Yaskawa INFORM job: FIGURE.JBI

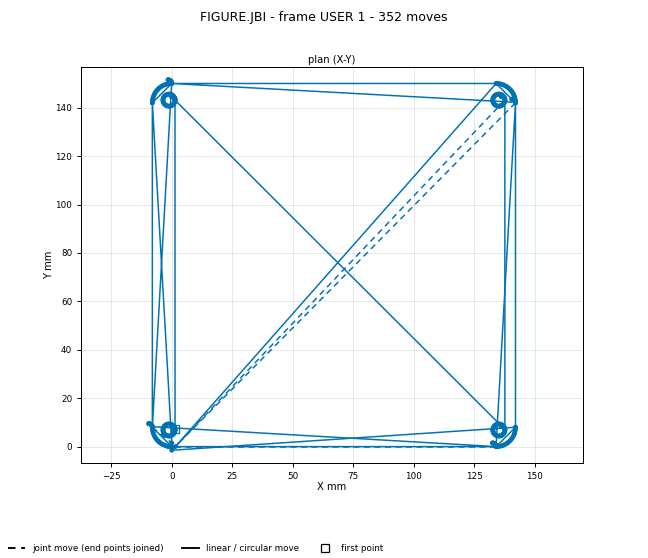
[picture p0: tool path of FIGURE.JBI in frame USER 1, 352 of 352 moves have a stored position in this frame; points joined in program order, loops and branches not executed]
/JOB
//NAME FIGURE
//POS
///NPOS 352,0,0,0,0,0
///TOOL 1
///USER 1
///POSTYPE USER
///RECTAN
///RCONF 1,0,0,0,0,0,0,0,0,0,0,0,0,0,0,0,0,0,0,0,0,0,0,0
C00000=1.357,7.11,7.0,0,0,0
C00001=1.302,7.339,7.0,0,0,0
C00002=1.212,7.556,7.0,0,0,0
C00003=1.089,7.757,7.0,0,0,0
C00004=0.936,7.936,7.0,0,0,0
C00005=0.757,8.089,7.0,0,0,0
C00006=0.556,8.212,7.0,0,0,0
C00007=0.339,8.302,7.0,0,0,0
C00008=0.11,8.357,7.0,0,0,0
C00009=-0.125,8.375,7.0,0,0,0
C00010=-0.125,8.375,7.0,0,0,0
C00011=1.375,6.875,7.0,0,0,0
C00012=1.344,7.266,7.0,0,0,0
C00013=1.253,7.648,7.0,0,0,0
C00014=1.103,8.01,7.0,0,0,0
C00015=0.898,8.344,7.0,0,0,0
C00016=0.643,8.643,7.0,0,0,0
C00017=0.344,8.898,7.0,0,0,0
C00018=0.01,9.103,7.0,0,0,0
C00019=-0.352,9.253,7.0,0,0,0
C00020=-0.734,9.344,7.0,0,0,0
C00021=-1.125,9.375,7.0,0,0,0
C00022=-1.516,9.344,7.0,0,0,0
C00023=-1.898,9.253,7.0,0,0,0
C00024=-2.26,9.103,7.0,0,0,0
C00025=-2.594,8.898,7.0,0,0,0
C00026=-2.893,8.643,7.0,0,0,0
C00027=-3.148,8.344,7.0,0,0,0
C00028=-3.353,8.01,7.0,0,0,0
C00029=-3.503,7.648,7.0,0,0,0
C00030=-3.594,7.266,7.0,0,0,0
C00031=-3.625,6.875,7.0,0,0,0
C00032=-3.594,6.484,7.0,0,0,0
C00033=-3.503,6.102,7.0,0,0,0
C00034=-3.353,5.74,7.0,0,0,0
C00035=-3.148,5.406,7.0,0,0,0
C00036=-2.893,5.107,7.0,0,0,0
C00037=-2.594,4.852,7.0,0,0,0
C00038=-2.26,4.647,7.0,0,0,0
C00039=-1.898,4.497,7.0,0,0,0
C00040=-1.516,4.406,7.0,0,0,0
C00041=-1.125,4.375,7.0,0,0,0
C00042=-0.734,4.406,7.0,0,0,0
C00043=-0.352,4.497,7.0,0,0,0
C00044=0.01,4.647,7.0,0,0,0
C00045=0.344,4.852,7.0,0,0,0
C00046=0.643,5.107,7.0,0,0,0
C00047=0.898,5.406,7.0,0,0,0
C00048=1.103,5.74,7.0,0,0,0
C00049=1.253,6.102,7.0,0,0,0
C00050=1.344,6.484,7.0,0,0,0
C00051=1.375,6.875,7.0,0,0,0
C00052=1.357,143.36,7.0,0,0,0
C00053=1.302,143.589,7.0,0,0,0
C00054=1.212,143.806,7.0,0,0,0
C00055=1.089,144.007,7.0,0,0,0
C00056=0.936,144.186,7.0,0,0,0
C00057=0.757,144.339,7.0,0,0,0
C00058=0.556,144.462,7.0,0,0,0
C00059=0.339,144.552,7.0,0,0,0
C00060=0.11,144.607,7.0,0,0,0
C00061=-0.125,144.625,7.0,0,0,0
C00062=-0.125,144.625,7.0,0,0,0
C00063=1.375,143.125,7.0,0,0,0
C00064=1.344,143.516,7.0,0,0,0
C00065=1.253,143.898,7.0,0,0,0
C00066=1.103,144.26,7.0,0,0,0
C00067=0.898,144.594,7.0,0,0,0
C00068=0.643,144.893,7.0,0,0,0
C00069=0.344,145.148,7.0,0,0,0
C00070=0.01,145.353,7.0,0,0,0
C00071=-0.352,145.503,7.0,0,0,0
C00072=-0.734,145.594,7.0,0,0,0
C00073=-1.125,145.625,7.0,0,0,0
C00074=-1.516,145.594,7.0,0,0,0
C00075=-1.898,145.503,7.0,0,0,0
C00076=-2.26,145.353,7.0,0,0,0
C00077=-2.594,145.148,7.0,0,0,0
C00078=-2.893,144.893,7.0,0,0,0
C00079=-3.148,144.594,7.0,0,0,0
C00080=-3.353,144.26,7.0,0,0,0
C00081=-3.503,143.898,7.0,0,0,0
C00082=-3.594,143.516,7.0,0,0,0
C00083=-3.625,143.125,7.0,0,0,0
C00084=-3.594,142.734,7.0,0,0,0
C00085=-3.503,142.352,7.0,0,0,0
C00086=-3.353,141.99,7.0,0,0,0
C00087=-3.148,141.656,7.0,0,0,0
C00088=-2.893,141.357,7.0,0,0,0
C00089=-2.594,141.102,7.0,0,0,0
C00090=-2.26,140.897,7.0,0,0,0
C00091=-1.898,140.747,7.0,0,0,0
C00092=-1.516,140.656,7.0,0,0,0
C00093=-1.125,140.625,7.0,0,0,0
C00094=-0.734,140.656,7.0,0,0,0
C00095=-0.352,140.747,7.0,0,0,0
C00096=0.01,140.897,7.0,0,0,0
C00097=0.344,141.102,7.0,0,0,0
C00098=0.643,141.357,7.0,0,0,0
C00099=0.898,141.656,7.0,0,0,0
C00100=1.103,141.99,7.0,0,0,0
C00101=1.253,142.352,7.0,0,0,0
C00102=1.344,142.734,7.0,0,0,0
C00103=1.375,143.125,7.0,0,0,0
C00104=137.607,7.11,7.0,0,0,0
C00105=137.552,7.339,7.0,0,0,0
C00106=137.462,7.556,7.0,0,0,0
C00107=137.339,7.757,7.0,0,0,0
C00108=137.186,7.936,7.0,0,0,0
C00109=137.007,8.089,7.0,0,0,0
C00110=136.806,8.212,7.0,0,0,0
C00111=136.589,8.302,7.0,0,0,0
C00112=136.36,8.357,7.0,0,0,0
C00113=136.125,8.375,7.0,0,0,0
C00114=136.125,8.375,7.0,0,0,0
C00115=137.625,6.875,7.0,0,0,0
C00116=137.594,7.266,7.0,0,0,0
C00117=137.503,7.648,7.0,0,0,0
C00118=137.353,8.01,7.0,0,0,0
C00119=137.148,8.344,7.0,0,0,0
C00120=136.893,8.643,7.0,0,0,0
C00121=136.594,8.898,7.0,0,0,0
C00122=136.26,9.103,7.0,0,0,0
C00123=135.898,9.253,7.0,0,0,0
C00124=135.516,9.344,7.0,0,0,0
C00125=135.125,9.375,7.0,0,0,0
C00126=134.734,9.344,7.0,0,0,0
C00127=134.352,9.253,7.0,0,0,0
C00128=133.99,9.103,7.0,0,0,0
C00129=133.656,8.898,7.0,0,0,0
C00130=133.357,8.643,7.0,0,0,0
C00131=133.102,8.344,7.0,0,0,0
C00132=132.897,8.01,7.0,0,0,0
C00133=132.747,7.648,7.0,0,0,0
C00134=132.656,7.266,7.0,0,0,0
C00135=132.625,6.875,7.0,0,0,0
C00136=132.656,6.484,7.0,0,0,0
C00137=132.747,6.102,7.0,0,0,0
C00138=132.897,5.74,7.0,0,0,0
C00139=133.102,5.406,7.0,0,0,0
C00140=133.357,5.107,7.0,0,0,0
C00141=133.656,4.852,7.0,0,0,0
C00142=133.99,4.647,7.0,0,0,0
C00143=134.352,4.497,7.0,0,0,0
C00144=134.734,4.406,7.0,0,0,0
C00145=135.125,4.375,7.0,0,0,0
C00146=135.516,4.406,7.0,0,0,0
C00147=135.898,4.497,7.0,0,0,0
C00148=136.26,4.647,7.0,0,0,0
C00149=136.594,4.852,7.0,0,0,0
C00150=136.893,5.107,7.0,0,0,0
C00151=137.148,5.406,7.0,0,0,0
C00152=137.353,5.74,7.0,0,0,0
C00153=137.503,6.102,7.0,0,0,0
C00154=137.594,6.484,7.0,0,0,0
C00155=137.625,6.875,7.0,0,0,0
C00156=137.607,143.36,7.0,0,0,0
C00157=137.552,143.589,7.0,0,0,0
C00158=137.462,143.806,7.0,0,0,0
C00159=137.339,144.007,7.0,0,0,0
C00160=137.186,144.186,7.0,0,0,0
C00161=137.007,144.339,7.0,0,0,0
C00162=136.806,144.462,7.0,0,0,0
C00163=136.589,144.552,7.0,0,0,0
C00164=136.36,144.607,7.0,0,0,0
C00165=136.125,144.625,7.0,0,0,0
C00166=136.125,144.625,7.0,0,0,0
C00167=137.625,143.125,7.0,0,0,0
C00168=137.594,143.516,7.0,0,0,0
C00169=137.503,143.898,7.0,0,0,0
C00170=137.353,144.26,7.0,0,0,0
C00171=137.148,144.594,7.0,0,0,0
C00172=136.893,144.893,7.0,0,0,0
C00173=136.594,145.148,7.0,0,0,0
C00174=136.26,145.353,7.0,0,0,0
C00175=135.898,145.503,7.0,0,0,0
C00176=135.516,145.594,7.0,0,0,0
C00177=135.125,145.625,7.0,0,0,0
C00178=134.734,145.594,7.0,0,0,0
C00179=134.352,145.503,7.0,0,0,0
C00180=133.99,145.353,7.0,0,0,0
C00181=133.656,145.148,7.0,0,0,0
C00182=133.357,144.893,7.0,0,0,0
C00183=133.102,144.594,7.0,0,0,0
C00184=132.897,144.26,7.0,0,0,0
C00185=132.747,143.898,7.0,0,0,0
C00186=132.656,143.516,7.0,0,0,0
C00187=132.625,143.125,7.0,0,0,0
C00188=132.656,142.734,7.0,0,0,0
C00189=132.747,142.352,7.0,0,0,0
C00190=132.897,141.99,7.0,0,0,0
C00191=133.102,141.656,7.0,0,0,0
C00192=133.357,141.357,7.0,0,0,0
C00193=133.656,141.102,7.0,0,0,0
C00194=133.99,140.897,7.0,0,0,0
C00195=134.352,140.747,7.0,0,0,0
C00196=134.734,140.656,7.0,0,0,0
C00197=135.125,140.625,7.0,0,0,0
C00198=135.516,140.656,7.0,0,0,0
C00199=135.898,140.747,7.0,0,0,0
C00200=136.26,140.897,7.0,0,0,0
C00201=136.594,141.102,7.0,0,0,0
C00202=136.893,141.357,7.0,0,0,0
C00203=137.148,141.656,7.0,0,0,0
C00204=137.353,141.99,7.0,0,0,0
C00205=137.503,142.352,7.0,0,0,0
C00206=137.594,142.734,7.0,0,0,0
C00207=137.625,143.125,7.0,0,0,0
C00208=1.5,-0.0,7.0,0,0,0
C00209=134.0,150.0,7.0,0,0,0
C00210=0.0,150.0,7.0,0,0,0
C00211=141.982,142.235,7.0,0,0,0
C00212=141.927,142.464,7.0,0,0,0
C00213=141.837,142.681,7.0,0,0,0
C00214=141.714,142.882,7.0,0,0,0
C00215=141.561,143.061,7.0,0,0,0
C00216=141.382,143.214,7.0,0,0,0
C00217=141.181,143.337,7.0,0,0,0
C00218=140.964,143.427,7.0,0,0,0
C00219=140.735,143.482,7.0,0,0,0
C00220=140.5,143.5,7.0,0,0,0
C00221=140.5,143.5,7.0,0,0,0
C00222=142.0,142.0,7.0,0,0,0
C00223=141.975,142.628,7.0,0,0,0
C00224=141.902,143.251,7.0,0,0,0
C00225=141.779,143.868,7.0,0,0,0
C00226=141.608,144.472,7.0,0,0,0
C00227=141.391,145.061,7.0,0,0,0
C00228=141.128,145.632,7.0,0,0,0
C00229=140.821,146.18,7.0,0,0,0
C00230=140.472,146.702,7.0,0,0,0
C00231=140.083,147.196,7.0,0,0,0
C00232=139.657,147.657,7.0,0,0,0
C00233=139.196,148.083,7.0,0,0,0
C00234=138.702,148.472,7.0,0,0,0
C00235=138.18,148.821,7.0,0,0,0
C00236=137.632,149.128,7.0,0,0,0
C00237=137.061,149.391,7.0,0,0,0
C00238=136.472,149.608,7.0,0,0,0
C00239=135.868,149.779,7.0,0,0,0
C00240=135.251,149.902,7.0,0,0,0
C00241=134.628,149.975,7.0,0,0,0
C00242=134.0,150.0,7.0,0,0,0
C00243=142.0,142.0,7.0,0,0,0
C00244=-0.0,-1.5,7.0,0,0,0
C00245=142.0,8.0,7.0,0,0,0
C00246=142.0,142.0,7.0,0,0,0
C00247=133.982,0.235,7.0,0,0,0
C00248=133.927,0.464,7.0,0,0,0
C00249=133.837,0.681,7.0,0,0,0
C00250=133.714,0.882,7.0,0,0,0
C00251=133.561,1.061,7.0,0,0,0
C00252=133.382,1.214,7.0,0,0,0
C00253=133.181,1.337,7.0,0,0,0
C00254=132.964,1.427,7.0,0,0,0
C00255=132.735,1.482,7.0,0,0,0
C00256=132.5,1.5,7.0,0,0,0
C00257=132.5,1.5,7.0,0,0,0
C00258=134.0,0.0,7.0,0,0,0
C00259=134.628,0.025,7.0,0,0,0
C00260=135.251,0.098,7.0,0,0,0
C00261=135.868,0.221,7.0,0,0,0
C00262=136.472,0.392,7.0,0,0,0
C00263=137.061,0.609,7.0,0,0,0
C00264=137.632,0.872,7.0,0,0,0
C00265=138.18,1.179,7.0,0,0,0
C00266=138.702,1.528,7.0,0,0,0
C00267=139.196,1.917,7.0,0,0,0
C00268=139.657,2.343,7.0,0,0,0
C00269=140.083,2.804,7.0,0,0,0
C00270=140.472,3.298,7.0,0,0,0
C00271=140.821,3.82,7.0,0,0,0
C00272=141.128,4.368,7.0,0,0,0
C00273=141.391,4.939,7.0,0,0,0
C00274=141.608,5.528,7.0,0,0,0
C00275=141.779,6.132,7.0,0,0,0
C00276=141.902,6.749,7.0,0,0,0
C00277=141.975,7.372,7.0,0,0,0
C00278=142.0,8.0,7.0,0,0,0
C00279=134.0,0.0,7.0,0,0,0
C00280=-1.5,-0.0,7.0,0,0,0
C00281=0.0,0.0,7.0,0,0,0
C00282=134.0,0.0,7.0,0,0,0
C00283=-8.018,8.235,7.0,0,0,0
C00284=-8.073,8.464,7.0,0,0,0
C00285=-8.163,8.681,7.0,0,0,0
C00286=-8.286,8.882,7.0,0,0,0
C00287=-8.439,9.061,7.0,0,0,0
C00288=-8.618,9.214,7.0,0,0,0
C00289=-8.819,9.337,7.0,0,0,0
C00290=-9.036,9.427,7.0,0,0,0
C00291=-9.265,9.482,7.0,0,0,0
C00292=-9.5,9.5,7.0,0,0,0
C00293=-9.5,9.5,7.0,0,0,0
C00294=-8.0,8.0,7.0,0,0,0
C00295=-7.975,7.372,7.0,0,0,0
C00296=-7.902,6.749,7.0,0,0,0
C00297=-7.779,6.132,7.0,0,0,0
C00298=-7.608,5.528,7.0,0,0,0
C00299=-7.391,4.939,7.0,0,0,0
C00300=-7.128,4.368,7.0,0,0,0
C00301=-6.821,3.82,7.0,0,0,0
C00302=-6.472,3.298,7.0,0,0,0
C00303=-6.083,2.804,7.0,0,0,0
C00304=-5.657,2.343,7.0,0,0,0
C00305=-5.196,1.917,7.0,0,0,0
C00306=-4.702,1.528,7.0,0,0,0
C00307=-4.18,1.179,7.0,0,0,0
C00308=-3.632,0.872,7.0,0,0,0
C00309=-3.061,0.609,7.0,0,0,0
C00310=-2.472,0.392,7.0,0,0,0
C00311=-1.868,0.221,7.0,0,0,0
C00312=-1.251,0.098,7.0,0,0,0
C00313=-0.628,0.025,7.0,0,0,0
C00314=-0.0,0.0,7.0,0,0,0
C00315=-8.0,8.0,7.0,0,0,0
C00316=0.0,1.5,7.0,0,0,0
C00317=-8.0,142.0,7.0,0,0,0
C00318=-8.0,8.0,7.0,0,0,0
C00319=-0.018,150.235,7.0,0,0,0
C00320=-0.073,150.464,7.0,0,0,0
C00321=-0.163,150.681,7.0,0,0,0
C00322=-0.286,150.882,7.0,0,0,0
C00323=-0.439,151.061,7.0,0,0,0
C00324=-0.618,151.214,7.0,0,0,0
C00325=-0.819,151.337,7.0,0,0,0
C00326=-1.036,151.427,7.0,0,0,0
C00327=-1.265,151.482,7.0,0,0,0
C00328=-1.5,151.5,7.0,0,0,0
C00329=-1.5,151.5,7.0,0,0,0
C00330=0.0,150.0,7.0,0,0,0
C00331=-0.628,149.975,7.0,0,0,0
C00332=-1.251,149.902,7.0,0,0,0
C00333=-1.868,149.779,7.0,0,0,0
C00334=-2.472,149.608,7.0,0,0,0
C00335=-3.061,149.391,7.0,0,0,0
C00336=-3.632,149.128,7.0,0,0,0
C00337=-4.18,148.821,7.0,0,0,0
C00338=-4.702,148.472,7.0,0,0,0
C00339=-5.196,148.083,7.0,0,0,0
C00340=-5.657,147.657,7.0,0,0,0
C00341=-6.083,147.196,7.0,0,0,0
C00342=-6.472,146.702,7.0,0,0,0
C00343=-6.821,146.18,7.0,0,0,0
C00344=-7.128,145.632,7.0,0,0,0
C00345=-7.391,145.061,7.0,0,0,0
C00346=-7.608,144.472,7.0,0,0,0
C00347=-7.779,143.868,7.0,0,0,0
C00348=-7.902,143.251,7.0,0,0,0
C00349=-7.975,142.628,7.0,0,0,0
C00350=-8.0,142.0,7.0,0,0,0
C00351=0.0,150.0,7.0,0,0,0
//INST
///DATE 2025/05/21 12:47
///ATTR SC,RW,RJ
////FRAME USER 1
///GROUP1 RB1
NOP
DOUT OT#(1) OFF
TIMER T=1.000
DOUT OT#(1) ON
TIMER T=1.000
DOUT OT#(1) OFF
TIMER T=1.000
DOUT OT#(1) ON
TIMER T=1.000
DOUT OT#(1) OFF
TIMER T=1.000
DOUT OT#(1) ON
TIMER T=1.000
DOUT OT#(1) OFF
TIMER T=1.000
DOUT OT#(1) ON
TIMER T=1.000
DOUT OT#(1) OFF
TIMER T=1.000
DOUT OT#(1) ON
TIMER T=1.000
DOUT OT#(1) OFF
TIMER T=1.000
DOUT OT#(1) ON
TIMER T=1.000
DOUT OT#(1) OFF
TIMER T=1.000
DOUT OT#(1) ON
TIMER T=1.000
DOUT OT#(1) OFF
TIMER T=1.000
DOUT OT#(1) ON
TIMER T=1.000
DOUT OT#(1) OFF
TIMER T=1.000
DOUT OT#(1) ON
TIMER T=1.000
DOUT OT#(1) OFF
TIMER T=1.000
DOUT OT#(1) ON
TIMER T=1.000
DOUT OT#(1) OFF
TIMER T=1.000
DOUT OT#(1) ON
TIMER T=1.000
DOUT OT#(1) OFF
TIMER T=1.000
DOUT OT#(1) ON
TIMER T=1.000
DOUT OT#(1) OFF
TIMER T=1.000
MOVL C00000 V=89 PL=0
MOVL C00001 V=89 PL=0
MOVL C00002 V=89 PL=0
MOVL C00003 V=89 PL=0
MOVL C00004 V=89 PL=0
MOVL C00005 V=89 PL=0
MOVL C00006 V=89 PL=0
MOVL C00007 V=89 PL=0
MOVL C00008 V=89 PL=0
MOVL C00009 V=89 PL=0
MOVJ C00010 VJ=30
MOVL C00011 V=89 PL=0
MOVL C00012 V=89 PL=0
MOVL C00013 V=89 PL=0
MOVL C00014 V=89 PL=0
MOVL C00015 V=89 PL=0
MOVL C00016 V=89 PL=0
MOVL C00017 V=89 PL=0
MOVL C00018 V=89 PL=0
MOVL C00019 V=89 PL=0
MOVL C00020 V=89 PL=0
MOVL C00021 V=89 PL=0
MOVL C00022 V=89 PL=0
MOVL C00023 V=89 PL=0
MOVL C00024 V=89 PL=0
MOVL C00025 V=89 PL=0
MOVL C00026 V=89 PL=0
MOVL C00027 V=89 PL=0
MOVL C00028 V=89 PL=0
MOVL C00029 V=89 PL=0
MOVL C00030 V=89 PL=0
MOVL C00031 V=89 PL=0
MOVL C00032 V=89 PL=0
MOVL C00033 V=89 PL=0
MOVL C00034 V=89 PL=0
MOVL C00035 V=89 PL=0
MOVL C00036 V=89 PL=0
MOVL C00037 V=89 PL=0
MOVL C00038 V=89 PL=0
MOVL C00039 V=89 PL=0
MOVL C00040 V=89 PL=0
MOVL C00041 V=89 PL=0
MOVL C00042 V=89 PL=0
MOVL C00043 V=89 PL=0
MOVL C00044 V=89 PL=0
MOVL C00045 V=89 PL=0
MOVL C00046 V=89 PL=0
MOVL C00047 V=89 PL=0
MOVL C00048 V=89 PL=0
MOVL C00049 V=89 PL=0
MOVL C00050 V=89 PL=0
MOVL C00051 V=89 PL=0
MOVL C00052 V=89 PL=0
MOVL C00053 V=89 PL=0
MOVL C00054 V=89 PL=0
MOVL C00055 V=89 PL=0
MOVL C00056 V=89 PL=0
MOVL C00057 V=89 PL=0
MOVL C00058 V=89 PL=0
MOVL C00059 V=89 PL=0
MOVL C00060 V=89 PL=0
MOVL C00061 V=89 PL=0
MOVJ C00062 VJ=30
MOVL C00063 V=89 PL=0
MOVL C00064 V=89 PL=0
MOVL C00065 V=89 PL=0
MOVL C00066 V=89 PL=0
MOVL C00067 V=89 PL=0
MOVL C00068 V=89 PL=0
MOVL C00069 V=89 PL=0
MOVL C00070 V=89 PL=0
MOVL C00071 V=89 PL=0
MOVL C00072 V=89 PL=0
MOVL C00073 V=89 PL=0
MOVL C00074 V=89 PL=0
MOVL C00075 V=89 PL=0
MOVL C00076 V=89 PL=0
MOVL C00077 V=89 PL=0
MOVL C00078 V=89 PL=0
MOVL C00079 V=89 PL=0
MOVL C00080 V=89 PL=0
MOVL C00081 V=89 PL=0
MOVL C00082 V=89 PL=0
MOVL C00083 V=89 PL=0
MOVL C00084 V=89 PL=0
MOVL C00085 V=89 PL=0
MOVL C00086 V=89 PL=0
MOVL C00087 V=89 PL=0
MOVL C00088 V=89 PL=0
MOVL C00089 V=89 PL=0
MOVL C00090 V=89 PL=0
MOVL C00091 V=89 PL=0
MOVL C00092 V=89 PL=0
MOVL C00093 V=89 PL=0
MOVL C00094 V=89 PL=0
MOVL C00095 V=89 PL=0
MOVL C00096 V=89 PL=0
MOVL C00097 V=89 PL=0
MOVL C00098 V=89 PL=0
MOVL C00099 V=89 PL=0
MOVL C00100 V=89 PL=0
MOVL C00101 V=89 PL=0
MOVL C00102 V=89 PL=0
MOVL C00103 V=89 PL=0
MOVL C00104 V=89 PL=0
MOVL C00105 V=89 PL=0
MOVL C00106 V=89 PL=0
MOVL C00107 V=89 PL=0
MOVL C00108 V=89 PL=0
MOVL C00109 V=89 PL=0
MOVL C00110 V=89 PL=0
MOVL C00111 V=89 PL=0
MOVL C00112 V=89 PL=0
MOVL C00113 V=89 PL=0
MOVJ C00114 VJ=30
MOVL C00115 V=89 PL=0
MOVL C00116 V=89 PL=0
MOVL C00117 V=89 PL=0
MOVL C00118 V=89 PL=0
MOVL C00119 V=89 PL=0
MOVL C00120 V=89 PL=0
MOVL C00121 V=89 PL=0
MOVL C00122 V=89 PL=0
MOVL C00123 V=89 PL=0
MOVL C00124 V=89 PL=0
MOVL C00125 V=89 PL=0
MOVL C00126 V=89 PL=0
MOVL C00127 V=89 PL=0
MOVL C00128 V=89 PL=0
MOVL C00129 V=89 PL=0
MOVL C00130 V=89 PL=0
MOVL C00131 V=89 PL=0
MOVL C00132 V=89 PL=0
MOVL C00133 V=89 PL=0
MOVL C00134 V=89 PL=0
MOVL C00135 V=89 PL=0
MOVL C00136 V=89 PL=0
MOVL C00137 V=89 PL=0
MOVL C00138 V=89 PL=0
MOVL C00139 V=89 PL=0
MOVL C00140 V=89 PL=0
MOVL C00141 V=89 PL=0
MOVL C00142 V=89 PL=0
MOVL C00143 V=89 PL=0
MOVL C00144 V=89 PL=0
MOVL C00145 V=89 PL=0
MOVL C00146 V=89 PL=0
MOVL C00147 V=89 PL=0
MOVL C00148 V=89 PL=0
MOVL C00149 V=89 PL=0
MOVL C00150 V=89 PL=0
MOVL C00151 V=89 PL=0
MOVL C00152 V=89 PL=0
MOVL C00153 V=89 PL=0
MOVL C00154 V=89 PL=0
MOVL C00155 V=89 PL=0
MOVL C00156 V=89 PL=0
MOVL C00157 V=89 PL=0
MOVL C00158 V=89 PL=0
MOVL C00159 V=89 PL=0
MOVL C00160 V=89 PL=0
MOVL C00161 V=89 PL=0
MOVL C00162 V=89 PL=0
MOVL C00163 V=89 PL=0
MOVL C00164 V=89 PL=0
MOVL C00165 V=89 PL=0
MOVJ C00166 VJ=30
MOVL C00167 V=89 PL=0
MOVL C00168 V=89 PL=0
MOVL C00169 V=89 PL=0
MOVL C00170 V=89 PL=0
MOVL C00171 V=89 PL=0
MOVL C00172 V=89 PL=0
MOVL C00173 V=89 PL=0
MOVL C00174 V=89 PL=0
MOVL C00175 V=89 PL=0
MOVL C00176 V=89 PL=0
MOVL C00177 V=89 PL=0
MOVL C00178 V=89 PL=0
MOVL C00179 V=89 PL=0
MOVL C00180 V=89 PL=0
MOVL C00181 V=89 PL=0
MOVL C00182 V=89 PL=0
MOVL C00183 V=89 PL=0
MOVL C00184 V=89 PL=0
MOVL C00185 V=89 PL=0
MOVL C00186 V=89 PL=0
MOVL C00187 V=89 PL=0
MOVL C00188 V=89 PL=0
MOVL C00189 V=89 PL=0
MOVL C00190 V=89 PL=0
MOVL C00191 V=89 PL=0
MOVL C00192 V=89 PL=0
MOVL C00193 V=89 PL=0
MOVL C00194 V=89 PL=0
MOVL C00195 V=89 PL=0
MOVL C00196 V=89 PL=0
MOVL C00197 V=89 PL=0
MOVL C00198 V=89 PL=0
MOVL C00199 V=89 PL=0
MOVL C00200 V=89 PL=0
MOVL C00201 V=89 PL=0
MOVL C00202 V=89 PL=0
MOVL C00203 V=89 PL=0
MOVL C00204 V=89 PL=0
MOVL C00205 V=89 PL=0
MOVL C00206 V=89 PL=0
MOVL C00207 V=89 PL=0
MOVJ C00208 VJ=30
MOVL C00209 V=89 PL=0
MOVL C00210 V=89 PL=0
MOVL C00211 V=89 PL=0
MOVL C00212 V=89 PL=0
MOVL C00213 V=89 PL=0
MOVL C00214 V=89 PL=0
MOVL C00215 V=89 PL=0
MOVL C00216 V=89 PL=0
MOVL C00217 V=89 PL=0
MOVL C00218 V=89 PL=0
MOVL C00219 V=89 PL=0
MOVL C00220 V=89 PL=0
MOVJ C00221 VJ=30
MOVL C00222 V=89 PL=0
MOVL C00223 V=89 PL=0
MOVL C00224 V=89 PL=0
MOVL C00225 V=89 PL=0
MOVL C00226 V=89 PL=0
MOVL C00227 V=89 PL=0
MOVL C00228 V=89 PL=0
MOVL C00229 V=89 PL=0
MOVL C00230 V=89 PL=0
MOVL C00231 V=89 PL=0
MOVL C00232 V=89 PL=0
MOVL C00233 V=89 PL=0
MOVL C00234 V=89 PL=0
MOVL C00235 V=89 PL=0
MOVL C00236 V=89 PL=0
MOVL C00237 V=89 PL=0
MOVL C00238 V=89 PL=0
MOVL C00239 V=89 PL=0
MOVL C00240 V=89 PL=0
MOVL C00241 V=89 PL=0
MOVL C00242 V=89 PL=0
MOVL C00243 V=89 PL=0
MOVJ C00244 VJ=30
MOVL C00245 V=89 PL=0
MOVL C00246 V=89 PL=0
MOVL C00247 V=89 PL=0
MOVL C00248 V=89 PL=0
MOVL C00249 V=89 PL=0
MOVL C00250 V=89 PL=0
MOVL C00251 V=89 PL=0
MOVL C00252 V=89 PL=0
MOVL C00253 V=89 PL=0
MOVL C00254 V=89 PL=0
MOVL C00255 V=89 PL=0
MOVL C00256 V=89 PL=0
MOVJ C00257 VJ=30
MOVL C00258 V=89 PL=0
MOVL C00259 V=89 PL=0
MOVL C00260 V=89 PL=0
MOVL C00261 V=89 PL=0
MOVL C00262 V=89 PL=0
MOVL C00263 V=89 PL=0
MOVL C00264 V=89 PL=0
MOVL C00265 V=89 PL=0
MOVL C00266 V=89 PL=0
MOVL C00267 V=89 PL=0
MOVL C00268 V=89 PL=0
MOVL C00269 V=89 PL=0
MOVL C00270 V=89 PL=0
MOVL C00271 V=89 PL=0
MOVL C00272 V=89 PL=0
MOVL C00273 V=89 PL=0
MOVL C00274 V=89 PL=0
MOVL C00275 V=89 PL=0
MOVL C00276 V=89 PL=0
MOVL C00277 V=89 PL=0
MOVL C00278 V=89 PL=0
MOVL C00279 V=89 PL=0
MOVJ C00280 VJ=30
MOVL C00281 V=89 PL=0
MOVL C00282 V=89 PL=0
MOVL C00283 V=89 PL=0
MOVL C00284 V=89 PL=0
MOVL C00285 V=89 PL=0
MOVL C00286 V=89 PL=0
MOVL C00287 V=89 PL=0
MOVL C00288 V=89 PL=0
MOVL C00289 V=89 PL=0
MOVL C00290 V=89 PL=0
MOVL C00291 V=89 PL=0
MOVL C00292 V=89 PL=0
MOVJ C00293 VJ=30
MOVL C00294 V=89 PL=0
MOVL C00295 V=89 PL=0
MOVL C00296 V=89 PL=0
MOVL C00297 V=89 PL=0
MOVL C00298 V=89 PL=0
MOVL C00299 V=89 PL=0
MOVL C00300 V=89 PL=0
MOVL C00301 V=89 PL=0
MOVL C00302 V=89 PL=0
MOVL C00303 V=89 PL=0
MOVL C00304 V=89 PL=0
MOVL C00305 V=89 PL=0
MOVL C00306 V=89 PL=0
MOVL C00307 V=89 PL=0
MOVL C00308 V=89 PL=0
MOVL C00309 V=89 PL=0
MOVL C00310 V=89 PL=0
MOVL C00311 V=89 PL=0
MOVL C00312 V=89 PL=0
MOVL C00313 V=89 PL=0
MOVL C00314 V=89 PL=0
MOVL C00315 V=89 PL=0
MOVJ C00316 VJ=30
MOVL C00317 V=89 PL=0
MOVL C00318 V=89 PL=0
MOVL C00319 V=89 PL=0
MOVL C00320 V=89 PL=0
MOVL C00321 V=89 PL=0
MOVL C00322 V=89 PL=0
MOVL C00323 V=89 PL=0
MOVL C00324 V=89 PL=0
MOVL C00325 V=89 PL=0
MOVL C00326 V=89 PL=0
MOVL C00327 V=89 PL=0
MOVL C00328 V=89 PL=0
MOVJ C00329 VJ=30
MOVL C00330 V=89 PL=0
MOVL C00331 V=89 PL=0
MOVL C00332 V=89 PL=0
MOVL C00333 V=89 PL=0
MOVL C00334 V=89 PL=0
MOVL C00335 V=89 PL=0
MOVL C00336 V=89 PL=0
MOVL C00337 V=89 PL=0
MOVL C00338 V=89 PL=0
MOVL C00339 V=89 PL=0
MOVL C00340 V=89 PL=0
MOVL C00341 V=89 PL=0
MOVL C00342 V=89 PL=0
MOVL C00343 V=89 PL=0
MOVL C00344 V=89 PL=0
MOVL C00345 V=89 PL=0
MOVL C00346 V=89 PL=0
MOVL C00347 V=89 PL=0
MOVL C00348 V=89 PL=0
MOVL C00349 V=89 PL=0
MOVL C00350 V=89 PL=0
MOVL C00351 V=89 PL=0
DOUT OT#(1) OFF
END
